// TIA Portal project "S7_1500_IO" (V18)

(* hardware
DEVICE "S7-1500/ET200MP-Station_1"  S7-1500 station
   slot 0: "Profilschiene_0"  Rack  6ES7 590-1***0-0AA0
   slot 1: "PLC_1"  CPU 1511-1 PN  6ES7 511-1AL03-0AB0  V3.0
      slot 3: "CPU-Display_1"  6ES7591-1AA00-0AA0
      slot 32768: "PROFINET-Schnittstelle_1"  X1
         slot 32769: "Port_1"  X1 P1
         slot 32770: "Port_2"  X1 P2
      slot 34817: "Virtual CP interface port_1"  Virtual CP interface port  Virtual CP interface port
DEVICE "GSD-Geraet_1"  GSD.Device.PN
   slot 0: "Baugruppenträger"  Rack  V1.0
   slot 0: "PN-Device"  CODESYS PROFINET Device  -  V4.5.0
      slot 0: "Submodule V1"  Submodule V1
      slot 1: "I"  I
         slot 1: "P1"  P1
   slot 1: "Input 8Bit_1"  Input 8Bit  -
      slot 0: "Submodule"  Submodule  -
   slot 2: "Output 8Bit_1"  Output 8Bit  -
      slot 0: "Submodule"  Submodule  -
   slot 3: "Input Float32_1"  Input Float32  -
      slot 0: "Submodule"  Submodule  -
   slot 4: "Output Float32_1"  Output Float32  -
      slot 0: "Submodule"  Submodule  -
*)

// ===== PLC "PLC_1"  CPU 1511-1 PN =====

VAR_GLOBAL   // PLC tag table "Standard-Variablentabelle"
   "InBit0" AT %I0.0 : Bool;
   "InBit1" AT %I0.1 : Bool;
   "OutBit0" AT %Q0.0 : Bool;
   "OutBit1" AT %Q0.1 : Bool;
   "InFloat1" AT %ID1 : Real;
   "OutFloat1" AT %QD1 : Real;
END_VAR

ORGANIZATION_BLOCK "Main"   // OB1, FBD, ProgramCycle
TITLE = "Main Program Sweep (Cycle)"
{ S7_Optimized_Access := 'TRUE' }
VERSION : 0.1
   VAR_INPUT
      Initial_Call : Bool;   // Initial call of this OB
      Remanence : Bool;   // =True, if remanent data are available
   END_VAR
BEGIN

REGION Network 1
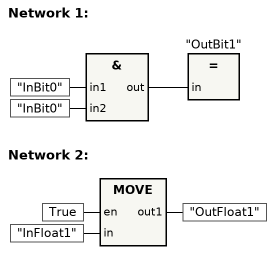
   "OutBit1" := "InBit0" AND "InBit0";
END_REGION

REGION Network 2
   IF True THEN "OutFloat1" := "InFloat1"; END_IF;
END_REGION
END_ORGANIZATION_BLOCK